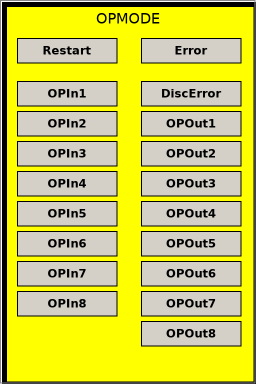
VISUALIZATION V_PH_OPMODE  // 256x384
VAR_INPUT
	stSafetyOPMODE			:ST_SAFETY_FBOPMODE;
END_VAR
    Rectangle (2,2 256x384), colour toggle: stSafetyOPMODE.bGeneralError
    Label (5,6 246x25), "OPMODE"
    RoundedRectangle (17,38 100x25), "Restart", colour toggle: stSafetyOPMODE.uStatus.stStatusWords.wInputs.0
    RoundedRectangle (17,81 100x25), "OPIn1", colour toggle: stSafetyOPMODE.uStatus.stStatusWords.wInputs.8
    RoundedRectangle (17,111 100x25), "OPIn2", colour toggle: stSafetyOPMODE.uStatus.stStatusWords.wInputs.9
    RoundedRectangle (17,201 100x25), "OPIn5", colour toggle: stSafetyOPMODE.uStatus.stStatusWords.wInputs.12
    RoundedRectangle (17,171 100x25), "OPIn4", colour toggle: stSafetyOPMODE.uStatus.stStatusWords.wInputs.11
    RoundedRectangle (17,141 100x25), "OPIn3", colour toggle: stSafetyOPMODE.uStatus.stStatusWords.wInputs.10
    RoundedRectangle (17,261 100x25), "OPIn7", colour toggle: stSafetyOPMODE.uStatus.stStatusWords.wInputs.14
    RoundedRectangle (17,291 100x25), "OPIn8", colour toggle: stSafetyOPMODE.uStatus.stStatusWords.wInputs.15
    RoundedRectangle (17,231 100x25), "OPIn6", colour toggle: stSafetyOPMODE.uStatus.stStatusWords.wInputs.13
    RoundedRectangle (141,81 100x25), "DiscError", colour toggle: stSafetyOPMODE.uStatus.stStatusWords.wDiagnosis.0, invisible if: NOT stSafetyOPMODE.uStatus.stStatusWords.wDiagnosis.0
    RoundedRectangle (141,38 100x25), "Error", colour toggle: stSafetyOPMODE.uStatus.stStatusWords.wOutputs.0
    RoundedRectangle (141,141 100x25), "OPOut2", colour toggle: stSafetyOPMODE.uStatus.stStatusWords.wOutputs.9
    RoundedRectangle (141,171 100x25), "OPOut3", colour toggle: stSafetyOPMODE.uStatus.stStatusWords.wOutputs.10
    RoundedRectangle (141,111 100x25), "OPOut1", colour toggle: stSafetyOPMODE.uStatus.stStatusWords.wOutputs.8
    RoundedRectangle (141,201 100x25), "OPOut4", colour toggle: stSafetyOPMODE.uStatus.stStatusWords.wOutputs.11
    RoundedRectangle (141,261 100x25), "OPOut6", colour toggle: stSafetyOPMODE.uStatus.stStatusWords.wOutputs.13
    RoundedRectangle (141,321 100x25), "OPOut8", colour toggle: stSafetyOPMODE.uStatus.stStatusWords.wOutputs.15
    RoundedRectangle (141,231 100x25), "OPOut5", colour toggle: stSafetyOPMODE.uStatus.stStatusWords.wOutputs.12
    RoundedRectangle (141,291 100x25), "OPOut7", colour toggle: stSafetyOPMODE.uStatus.stStatusWords.wOutputs.14
    Textfield (17,354 234x25), text list: 'TL_FbState', text index: stSafetyOPMODE.eState
END_VISUALIZATION

(* stored: Version 1.1.0.1, ProductVersion 3.1.4024.4
   Visu V_PH_OPMODE: Id {ce1ee3d6-9de9-448a-ab68-a63660fd085d} *)
